// FICTIONAL ENGINEERING PROJECT — NOT FOR CONSTRUCTION
FUNCTION_BLOCK "FB_CellMain"
VAR
   HmiCommands : "FB_HMICommandManager";
   ConveyorVfd : "FB_VFD";
   PumpVfd : "FB_VFD";
   Gate : "FB_Actuator2Pos";
   Clamp : "FB_Actuator2Pos";
   FillCh1 : "FB_FillChannel";
   FillCh2 : "FB_FillChannel";
   Vision : "FB_VisionInterface";
   Capper : "FB_CapperInterface";
   Recipe : "FB_RecipeManager";
   Alarm : "FB_AlarmManager";
   Coordinator : "FB_MachineCoordinator";
   DripTimer : TON;
   PlcHeartbeatTimer : TON;
   blockingFault : Bool;
   outputInterlock : Bool;
   preBlockingFault : Bool;
   immediateStop : Bool;
   processPermissive : Bool;
   modelConfigured : Bool;
   visionOperational : Bool;
   manualConveyorInterlocked : Bool;
   manualSecureInterlocked : Bool;
   manualPumpInterlocked : Bool;
   manualValve1Interlocked : Bool;
   manualValve2Interlocked : Bool;
   activeFaults : Array[0..31] of Bool;
   faultCodes : Array[0..31] of UInt;
   i : Int;
END_VAR
BEGIN
   // Input normalization from process image.
   "DB_IO".Inputs.SafetyOk := %I0.0;
   "DB_IO".Inputs.GuardClosed := %I0.1;
   "DB_IO".Inputs.AirPressureOk := %I0.2;
   "DB_IO".Inputs.ProductSupplyOk := %I0.3;
   "DB_IO".Inputs.Bottle1Present := %I1.2;
   "DB_IO".Inputs.Bottle2Present := %I1.3;
   "DB_IO".Inputs.GateOpen := %I1.4;
   "DB_IO".Inputs.GateClosed := %I1.5;
   "DB_IO".Inputs.ClampReleased := %I1.6;
   "DB_IO".Inputs.ClampEngaged := %I1.7;
   "DB_IO".Inputs.Valve1Closed := %I2.0;
   "DB_IO".Inputs.Valve2Closed := %I2.1;
   "DB_IO".Inputs.CapperReady := %I2.2;
   "DB_IO".Inputs.CapperBusy := %I2.3;
   "DB_IO".Inputs.CapperComplete := %I2.4;
   "DB_IO".Inputs.CapperFault := %I2.5;
   "DB_IO".Inputs.LocalReset := %I2.6;
   "DB_IO".Inputs.LocalStop := %I2.7;
   "DB_IO".Inputs.Flow1Raw := %IW64;
   "DB_IO".Inputs.Flow2Raw := %IW66;
   // Native-project adapter contract. Bind these fields to PN diagnostics and TM Count technology-object outputs in TIA V20.
   "DB_IO".Inputs.ConveyorPnHealthy := "DB_NativeBindings".Inputs.ConveyorPnIoValid;
   "DB_IO".Inputs.PumpPnHealthy := "DB_NativeBindings".Inputs.PumpPnIoValid;
   "DB_IO".Inputs.PulseTotal1 := "DB_NativeBindings".Inputs.Flow1PulseTotal;
   "DB_IO".Inputs.PulseTotal2 := "DB_NativeBindings".Inputs.Flow2PulseTotal;
   "DB_IO".Inputs.Flow1ChannelFault := "DB_NativeBindings".Inputs.Flow1ChannelFault;
   "DB_IO".Inputs.Flow2ChannelFault := "DB_NativeBindings".Inputs.Flow2ChannelFault;
   "DB_IO".Inputs.Flow1PulseChannelFault := "DB_NativeBindings".Inputs.Flow1PulseChannelFault;
   "DB_IO".Inputs.Flow2PulseChannelFault := "DB_NativeBindings".Inputs.Flow2PulseChannelFault;
   "DB_Drives".Conveyor.StatusWord1 := %IW256;
   "DB_Drives".Conveyor.ActualSpeedPzd := %IW258;
   "DB_Drives".Pump.StatusWord1 := %IW260;
   "DB_Drives".Pump.ActualSpeedPzd := %IW262;

   #modelConfigured := "DB_VisionComms".ModelConfigurationApproved AND ("DB_VisionComms".ExpectedModelId <> '') AND (LEN("DB_VisionComms".ExpectedModelHash) = 64)
      AND ("DB_VisionComms".ExpectedDatasetId <> '') AND ("DB_VisionComms".ExpectedCalibrationId <> '')
      AND ("DB_VisionComms".MinimumConfidence > 0.0) AND ("DB_VisionComms".MinimumConfidence <= 1.0)
      AND ("DB_VisionComms".MaximumResultAgeMs > UDINT#0) AND ("DB_VisionComms".MaximumProcessingTimeMs > UDINT#0);
   #visionOperational := "DB_VisionComms".Ready AND "DB_VisionComms".ServiceHealthy AND "DB_VisionComms".CameraHealthy
      AND "DB_VisionComms".ModelLoaded AND NOT "DB_VisionComms".MaintenanceActive;
   #immediateStop := NOT "DB_IO".Inputs.SafetyOk OR NOT "DB_IO".Inputs.GuardClosed OR NOT "DB_IO".Inputs.AirPressureOk OR NOT "DB_IO".Inputs.ProductSupplyOk;
   #processPermissive := NOT #immediateStop AND NOT "DB_IO".PowerRecoveryRequired;
   #preBlockingFault := #immediateStop OR #ConveyorVfd.Fault OR #PumpVfd.Fault OR #Gate.Fault OR #Clamp.Fault OR #FillCh1.Fault OR #FillCh2.Fault OR #Vision.Fault OR NOT #modelConfigured OR NOT #visionOperational OR #Capper.Fault OR NOT #HmiCommands.CommunicationsHealthy;
   #HmiCommands(StartRequest := "DB_HMI".Start.Request, StartSeq := "DB_HMI".Start.RequestSeq, StopRequest := "DB_HMI".ControlledStop.Request, StopSeq := "DB_HMI".ControlledStop.RequestSeq, ResetRequest := "DB_HMI".Reset.Request, ResetSeq := "DB_HMI".Reset.RequestSeq, AckRequest := "DB_HMI".AlarmAck.Request, AckSeq := "DB_HMI".AlarmAck.RequestSeq, AutoRequest := "DB_HMI".AutoMode.Request, AutoSeq := "DB_HMI".AutoMode.RequestSeq, ManualRequest := "DB_HMI".ManualMode.Request, ManualSeq := "DB_HMI".ManualMode.RequestSeq, DispositionRequest := "DB_HMI".DispositionRemoved.Request, DispositionSeq := "DB_HMI".DispositionRemoved.RequestSeq, ManualConveyorRequest := "DB_HMI".ManualConveyorJog.Request, ManualPumpRequest := "DB_HMI".ManualPumpJog.Request, ManualValve1Request := "DB_HMI".ManualValve1.Request, ManualValve2Request := "DB_HMI".ManualValve2.Request, ManualSecureRequest := "DB_HMI".ManualSecure.Request, ManualHoldAllowed := (#Coordinator.State = "E_MachineState".MANUAL_SETUP) AND #processPermissive, LocalStop := "DB_IO".Inputs.LocalStop, LocalReset := "DB_IO".Inputs.LocalReset, CommandHeartbeat := "DB_HMI".CommandHeartbeat, StartAllowed := (#Coordinator.State = "E_MachineState".READY) AND #processPermissive, ResetAllowed := NOT #immediateStop, AutoAllowed := (#Coordinator.State = "E_MachineState".MANUAL_SETUP), ManualAllowed := (#Coordinator.State = "E_MachineState".READY), DispositionAllowed := (#Coordinator.State = "E_MachineState".HOLDING));
   "DB_HMI".Start.AcceptedSeq := #HmiCommands.StartAcceptedSeq; "DB_HMI".Start.RejectedSeq := #HmiCommands.StartRejectedSeq;
   "DB_HMI".ControlledStop.AcceptedSeq := #HmiCommands.StopAcceptedSeq;
   "DB_HMI".Reset.AcceptedSeq := #HmiCommands.ResetAcceptedSeq; "DB_HMI".Reset.RejectedSeq := #HmiCommands.ResetRejectedSeq;
   "DB_HMI".AlarmAck.AcceptedSeq := #HmiCommands.AckAcceptedSeq;
   "DB_HMI".AutoMode.AcceptedSeq := #HmiCommands.AutoAcceptedSeq; "DB_HMI".AutoMode.RejectedSeq := #HmiCommands.AutoRejectedSeq;
   "DB_HMI".ManualMode.AcceptedSeq := #HmiCommands.ManualAcceptedSeq; "DB_HMI".ManualMode.RejectedSeq := #HmiCommands.ManualRejectedSeq;
   "DB_HMI".DispositionRemoved.AcceptedSeq := #HmiCommands.DispositionAcceptedSeq; "DB_HMI".DispositionRemoved.RejectedSeq := #HmiCommands.DispositionRejectedSeq;
   "DB_HMI".CommunicationsHealthy := #HmiCommands.CommunicationsHealthy;
   #manualConveyorInterlocked := #HmiCommands.ManualConveyorCmd AND NOT #HmiCommands.ManualSecureCmd AND NOT #HmiCommands.ManualPumpCmd AND NOT #HmiCommands.ManualValve1Cmd AND NOT #HmiCommands.ManualValve2Cmd AND "DB_IO".Inputs.GateOpen AND "DB_IO".Inputs.ClampReleased;
   #manualSecureInterlocked := #HmiCommands.ManualSecureCmd AND NOT #HmiCommands.ManualConveyorCmd AND #ConveyorVfd.Stopped;
   #manualPumpInterlocked := #HmiCommands.ManualPumpCmd AND #manualSecureInterlocked AND #ConveyorVfd.Stopped AND "DB_IO".Inputs.GateClosed AND "DB_IO".Inputs.ClampEngaged AND (#HmiCommands.ManualValve1Cmd OR #HmiCommands.ManualValve2Cmd);
   #manualValve1Interlocked := #HmiCommands.ManualValve1Cmd AND #manualPumpInterlocked AND #PumpVfd.Running;
   #manualValve2Interlocked := #HmiCommands.ManualValve2Cmd AND #manualPumpInterlocked AND #PumpVfd.Running;
   "DB_HMI".Start.Allowed := (#Coordinator.State = "E_MachineState".READY) AND #processPermissive; "DB_HMI".Start.Busy := FALSE; "DB_HMI".Start.DisabledReason := 0; IF NOT "DB_HMI".Start.Allowed THEN "DB_HMI".Start.DisabledReason := 1; END_IF;
   "DB_HMI".ControlledStop.Allowed := TRUE; "DB_HMI".ControlledStop.Busy := FALSE; "DB_HMI".ControlledStop.DisabledReason := 0;
   "DB_HMI".Reset.Allowed := NOT #immediateStop; "DB_HMI".Reset.Busy := FALSE; "DB_HMI".Reset.DisabledReason := 0; IF NOT "DB_HMI".Reset.Allowed THEN "DB_HMI".Reset.DisabledReason := 2; END_IF;
   "DB_HMI".AlarmAck.Allowed := TRUE; "DB_HMI".AlarmAck.Busy := FALSE; "DB_HMI".AlarmAck.DisabledReason := 0;
   "DB_HMI".AutoMode.Allowed := (#Coordinator.State = "E_MachineState".MANUAL_SETUP); "DB_HMI".AutoMode.Busy := FALSE; "DB_HMI".AutoMode.DisabledReason := 0; IF NOT "DB_HMI".AutoMode.Allowed THEN "DB_HMI".AutoMode.DisabledReason := 4; END_IF;
   "DB_HMI".ManualMode.Allowed := (#Coordinator.State = "E_MachineState".READY); "DB_HMI".ManualMode.Busy := FALSE; "DB_HMI".ManualMode.DisabledReason := 0; IF NOT "DB_HMI".ManualMode.Allowed THEN "DB_HMI".ManualMode.DisabledReason := 4; END_IF;
   "DB_HMI".DispositionRemoved.Allowed := (#Coordinator.State = "E_MachineState".HOLDING); "DB_HMI".DispositionRemoved.Busy := FALSE; "DB_HMI".DispositionRemoved.DisabledReason := 0;
   "DB_HMI".ManualConveyorJog.Allowed := (#Coordinator.State = "E_MachineState".MANUAL_SETUP) AND #processPermissive AND NOT #HmiCommands.ManualSecureCmd AND NOT #HmiCommands.ManualPumpCmd AND NOT #HmiCommands.ManualValve1Cmd AND NOT #HmiCommands.ManualValve2Cmd AND "DB_IO".Inputs.GateOpen AND "DB_IO".Inputs.ClampReleased; "DB_HMI".ManualConveyorJog.Busy := #manualConveyorInterlocked; "DB_HMI".ManualConveyorJog.DisabledReason := 0; IF NOT "DB_HMI".ManualConveyorJog.Allowed THEN "DB_HMI".ManualConveyorJog.DisabledReason := 5; END_IF;
   "DB_HMI".ManualPumpJog.Allowed := (#Coordinator.State = "E_MachineState".MANUAL_SETUP) AND #processPermissive AND #manualSecureInterlocked AND #ConveyorVfd.Stopped AND "DB_IO".Inputs.GateClosed AND "DB_IO".Inputs.ClampEngaged; "DB_HMI".ManualPumpJog.Busy := #manualPumpInterlocked; "DB_HMI".ManualPumpJog.DisabledReason := 0; IF NOT "DB_HMI".ManualPumpJog.Allowed THEN "DB_HMI".ManualPumpJog.DisabledReason := 6; END_IF;
   "DB_HMI".ManualValve1.Allowed := "DB_HMI".ManualPumpJog.Allowed; "DB_HMI".ManualValve1.Busy := #manualValve1Interlocked; "DB_HMI".ManualValve1.DisabledReason := "DB_HMI".ManualPumpJog.DisabledReason;
   "DB_HMI".ManualValve2.Allowed := "DB_HMI".ManualPumpJog.Allowed; "DB_HMI".ManualValve2.Busy := #manualValve2Interlocked; "DB_HMI".ManualValve2.DisabledReason := "DB_HMI".ManualPumpJog.DisabledReason;
   "DB_HMI".ManualSecure.Allowed := (#Coordinator.State = "E_MachineState".MANUAL_SETUP) AND #processPermissive AND #ConveyorVfd.Stopped AND NOT #HmiCommands.ManualConveyorCmd; "DB_HMI".ManualSecure.Busy := #manualSecureInterlocked; "DB_HMI".ManualSecure.DisabledReason := 0; IF NOT "DB_HMI".ManualSecure.Allowed THEN "DB_HMI".ManualSecure.DisabledReason := 7; END_IF;

   #Recipe(Candidate := "DB_Recipe".Candidate, ApplyRequest := "DB_HMI".RecipeApply.Request AND #HmiCommands.CommunicationsHealthy, RequestSeq := "DB_HMI".RecipeApply.RequestSeq, MachineStopped := (#Coordinator.State = "E_MachineState".STOPPED));
   "DB_Recipe".Active := #Recipe.Active;
   "DB_HMI".RecipeApply.AcceptedSeq := #Recipe.AcceptedSeq; "DB_HMI".RecipeApply.RejectedSeq := #Recipe.RejectedSeq;
   "DB_HMI".RecipeApply.Allowed := (#Coordinator.State = "E_MachineState".STOPPED) AND #Recipe.Valid; "DB_HMI".RecipeApply.Busy := FALSE; "DB_HMI".RecipeApply.DisabledReason := 0; IF NOT #Recipe.Valid THEN "DB_HMI".RecipeApply.DisabledReason := 3; END_IF;

   "DB_Drives".Conveyor.CommsHealthy := "DB_IO".Inputs.ConveyorPnHealthy; "DB_Drives".Pump.CommsHealthy := "DB_IO".Inputs.PumpPnHealthy;
   #ConveyorVfd(Enable := "DB_IO".Inputs.SafetyOk AND "DB_IO".Inputs.GuardClosed, RunRequest := (#Coordinator.IndexRequest OR #manualConveyorInterlocked) AND NOT #immediateStop, ResetEdge := #HmiCommands.ResetPulse, CommsHealthy := "DB_Drives".Conveyor.CommsHealthy, StatusWord1 := "DB_Drives".Conveyor.StatusWord1, ActualSpeedPzd := "DB_Drives".Conveyor.ActualSpeedPzd, SpeedReferencePct := 35.0, StartTimeout := T#3s, StopTimeout := T#3s);
   #PumpVfd(Enable := #processPermissive, RunRequest := ((#FillCh1.PumpRequest OR #FillCh2.PumpRequest) OR #manualPumpInterlocked) AND #processPermissive, ResetEdge := #HmiCommands.ResetPulse, CommsHealthy := "DB_Drives".Pump.CommsHealthy, StatusWord1 := "DB_Drives".Pump.StatusWord1, ActualSpeedPzd := "DB_Drives".Pump.ActualSpeedPzd, SpeedReferencePct := 60.0, StartTimeout := T#3s, StopTimeout := T#3s);
   "DB_Drives".Conveyor.Ready := #ConveyorVfd.Ready; "DB_Drives".Conveyor.Running := #ConveyorVfd.Running; "DB_Drives".Conveyor.Fault := #ConveyorVfd.Fault; "DB_Drives".Conveyor.ActualSpeedPct := #ConveyorVfd.ActualSpeedPct;
   "DB_Drives".Pump.Ready := #PumpVfd.Ready; "DB_Drives".Pump.Running := #PumpVfd.Running; "DB_Drives".Pump.Fault := #PumpVfd.Fault; "DB_Drives".Pump.ActualSpeedPct := #PumpVfd.ActualSpeedPct;
   #Gate(Enable := NOT #immediateStop, CmdToA := NOT (#Coordinator.GateCloseRequest OR #manualSecureInterlocked), CmdToB := #Coordinator.GateCloseRequest OR #manualSecureInterlocked, AtA := "DB_IO".Inputs.GateOpen, AtB := "DB_IO".Inputs.GateClosed, ResetEdge := #HmiCommands.ResetPulse, TravelTime := T#2s);
   #Clamp(Enable := NOT #immediateStop, CmdToA := NOT (#Coordinator.ClampRequest OR #manualSecureInterlocked), CmdToB := #Coordinator.ClampRequest OR #manualSecureInterlocked, AtA := "DB_IO".Inputs.ClampReleased, AtB := "DB_IO".Inputs.ClampEngaged, ResetEdge := #HmiCommands.ResetPulse, TravelTime := T#2s);
   #FillCh1(Enable := #processPermissive, PumpRunning := #PumpVfd.Running, StartEdge := #Coordinator.FillStartPulse, Abort := #preBlockingFault OR #ConveyorVfd.Fault OR #PumpVfd.Fault OR #Gate.Fault OR #Clamp.Fault OR #HmiCommands.StopPulse, ResetEdge := #HmiCommands.ResetPulse, PulseTotal := "DB_IO".Inputs.PulseTotal1, FlowRaw := "DB_IO".Inputs.Flow1Raw, PulseChannelFault := "DB_IO".Inputs.Flow1PulseChannelFault, AnalogChannelFault := "DB_IO".Inputs.Flow1ChannelFault, ValveClosedFb := "DB_IO".Inputs.Valve1Closed, TargetMl := "DB_Recipe".Active.TargetMlCh1, PulsesPerLitre := "DB_Recipe".Active.PulsesPerLitreCh1, UnderToleranceMl := "DB_Recipe".Active.UnderToleranceMl, OverToleranceMl := "DB_Recipe".Active.OverToleranceMl, FlowMaxLMin := 20.0, NoFlowMinLMin := 0.2, PlausibilityPct := 25.0, PulseWindowTimeS := "DB_Recipe".Active.PulseWindowTimeS, NoFlowTimeout := "DB_Recipe".Active.NoFlowTimeout, FillTimeout := "DB_Recipe".Active.FillTimeout, ValveOpenTimeout := "DB_Recipe".Active.ValveOpenTimeout, ValveCloseTimeout := "DB_Recipe".Active.ValveCloseTimeout, PlausibilityTime := "DB_Recipe".Active.PlausibilityTime);
   #FillCh2(Enable := #processPermissive, PumpRunning := #PumpVfd.Running, StartEdge := #Coordinator.FillStartPulse, Abort := #preBlockingFault OR #ConveyorVfd.Fault OR #PumpVfd.Fault OR #Gate.Fault OR #Clamp.Fault OR #HmiCommands.StopPulse, ResetEdge := #HmiCommands.ResetPulse, PulseTotal := "DB_IO".Inputs.PulseTotal2, FlowRaw := "DB_IO".Inputs.Flow2Raw, PulseChannelFault := "DB_IO".Inputs.Flow2PulseChannelFault, AnalogChannelFault := "DB_IO".Inputs.Flow2ChannelFault, ValveClosedFb := "DB_IO".Inputs.Valve2Closed, TargetMl := "DB_Recipe".Active.TargetMlCh2, PulsesPerLitre := "DB_Recipe".Active.PulsesPerLitreCh2, UnderToleranceMl := "DB_Recipe".Active.UnderToleranceMl, OverToleranceMl := "DB_Recipe".Active.OverToleranceMl, FlowMaxLMin := 20.0, NoFlowMinLMin := 0.2, PlausibilityPct := 25.0, PulseWindowTimeS := "DB_Recipe".Active.PulseWindowTimeS, NoFlowTimeout := "DB_Recipe".Active.NoFlowTimeout, FillTimeout := "DB_Recipe".Active.FillTimeout, ValveOpenTimeout := "DB_Recipe".Active.ValveOpenTimeout, ValveCloseTimeout := "DB_Recipe".Active.ValveCloseTimeout, PlausibilityTime := "DB_Recipe".Active.PlausibilityTime);
   #DripTimer(IN := (#Coordinator.AutoStep = "E_AutoStep".DRIP_SETTLE), PT := "DB_Recipe".Active.DripSettleTime);
   #Capper(Enable := NOT #immediateStop, RequestEdge := #Coordinator.CapperRequestPulse, Ready := "DB_IO".Inputs.CapperReady, Busy := "DB_IO".Inputs.CapperBusy, Complete := "DB_IO".Inputs.CapperComplete, FaultIn := "DB_IO".Inputs.CapperFault, ResetEdge := #HmiCommands.ResetPulse, AcceptTimeout := T#2s, CompleteTimeout := T#10s);
   // Allocate exactly one immutable ID. A repeated coordinator pulse cannot mutate
   // the externally visible transaction while the vision interface is pending.
   IF #Coordinator.VisionRequestPulse AND NOT #Vision.RequestInProgress AND ("DB_VisionComms".InspectionId < UDINT#4294967295) THEN "DB_VisionComms".InspectionId := "DB_VisionComms".InspectionId + UDINT#1; END_IF;
   // READY low holds VISION_ENABLE low so a cold/restarted edge can atomically
   // seed the PLC session/ID/ACK/heartbeat snapshot before declaring READY.
   "DB_VisionComms".MaintenanceMode := (#Coordinator.State = "E_MachineState".MANUAL_SETUP);
   "DB_VisionComms".Enable := #processPermissive AND #modelConfigured AND "DB_VisionComms".Ready AND #visionOperational
      AND NOT "DB_VisionComms".MaintenanceMode AND NOT #Vision.Fault;
   "DB_VisionComms".RecipeId := "DB_Recipe".Active.RecipeId; "DB_VisionComms".ExpectedBottles := 2; "DB_VisionComms".TargetFillLevel := "DB_Recipe".Active.TargetFillLevel;
   #PlcHeartbeatTimer(IN := NOT #PlcHeartbeatTimer.Q, PT := T#500ms);
   IF #PlcHeartbeatTimer.Q THEN
      IF "DB_VisionComms".PlcHeartbeat = UDINT#4294967295 THEN "DB_VisionComms".PlcHeartbeat := UDINT#0;
      ELSE "DB_VisionComms".PlcHeartbeat := "DB_VisionComms".PlcHeartbeat + UDINT#1; END_IF;
   END_IF;
   #Vision(Enable := "DB_VisionComms".Enable, TriggerEdge := #Coordinator.VisionRequestPulse,
      InspectionId := "DB_VisionComms".InspectionId, SessionEpoch := "DB_VisionComms".SessionEpoch,
      ExpectedModelId := "DB_VisionComms".ExpectedModelId, ExpectedModelHash := "DB_VisionComms".ExpectedModelHash,
      ExpectedDatasetId := "DB_VisionComms".ExpectedDatasetId, ExpectedCalibrationId := "DB_VisionComms".ExpectedCalibrationId,
      MinimumConfidence := "DB_VisionComms".MinimumConfidence, MaximumResultAgeMs := "DB_VisionComms".MaximumResultAgeMs,
      MaximumProcessingTimeMs := "DB_VisionComms".MaximumProcessingTimeMs, MaximumQueueDepth := "DB_VisionComms".MaximumQueueDepth,
      Ready := "DB_VisionComms".Ready, Busy := "DB_VisionComms".Busy, CaptureAckId := "DB_VisionComms".CaptureAckId,
      ProcessingState := "DB_VisionComms".ProcessingState, ServiceHealthy := "DB_VisionComms".ServiceHealthy,
      CameraHealthy := "DB_VisionComms".CameraHealthy, ModelLoaded := "DB_VisionComms".ModelLoaded,
      MaintenanceActive := "DB_VisionComms".MaintenanceActive, QueueDepth := "DB_VisionComms".QueueDepth,
      Result := "DB_VisionComms".Result, Heartbeat := "DB_VisionComms".VisionHeartbeat,
      Timeout := "DB_Recipe".Active.VisionTimeout, HeartbeatTimeout := T#1s, ResetEdge := #HmiCommands.ResetPulse);
   "DB_VisionComms".Trigger := #Vision.Trigger;
   "DB_VisionComms".ResultAgeMs := #Vision.ResultAgeMs;
   IF NOT #modelConfigured THEN "DB_VisionComms".DiagReason := "E_VisionDiag".MODEL_MISMATCH;
   ELSIF NOT "DB_VisionComms".ServiceHealthy THEN "DB_VisionComms".DiagReason := "E_VisionDiag".SERVICE_UNHEALTHY;
   ELSIF NOT "DB_VisionComms".CameraHealthy THEN "DB_VisionComms".DiagReason := "E_VisionDiag".CAMERA_UNHEALTHY;
   ELSIF NOT "DB_VisionComms".ModelLoaded THEN "DB_VisionComms".DiagReason := "E_VisionDiag".MODEL_NOT_LOADED;
   ELSIF "DB_VisionComms".MaintenanceActive THEN "DB_VisionComms".DiagReason := "E_VisionDiag".MAINTENANCE_ACTIVE;
   ELSE "DB_VisionComms".DiagReason := #Vision.DiagReason; END_IF;
   IF #Vision.PublicationAck THEN "DB_VisionComms".ResultAckId := "DB_VisionComms".Result.ResultId; END_IF;
   FOR #i := 0 TO 31 DO #activeFaults[#i] := FALSE; #faultCodes[#i] := 0; END_FOR;
   #activeFaults[0] := NOT "DB_IO".Inputs.SafetyOk; #faultCodes[0] := 1001;
   #activeFaults[1] := NOT "DB_IO".Inputs.GuardClosed; #faultCodes[1] := 1004;
   #activeFaults[2] := NOT "DB_IO".Inputs.AirPressureOk; #faultCodes[2] := 1002;
   #activeFaults[3] := NOT "DB_IO".Inputs.ProductSupplyOk; #faultCodes[3] := 1003;
   #activeFaults[4] := #ConveyorVfd.Fault; #faultCodes[4] := 1101;
   #activeFaults[5] := #PumpVfd.Fault; #faultCodes[5] := 1102;
   #activeFaults[6] := #Gate.Fault; #faultCodes[6] := 1201;
   #activeFaults[7] := #Clamp.Fault; #faultCodes[7] := 1202;
   #activeFaults[8] := #FillCh1.Fault; CASE #FillCh1.DiagReason OF "E_FillDiag".ANALOG_BROKEN_WIRE: #faultCodes[8] := 1307; "E_FillDiag".NO_FLOW: #faultCodes[8] := 1301; "E_FillDiag".PULSE_MISSING: #faultCodes[8] := 1321; "E_FillDiag".ANALOG_NO_FLOW: #faultCodes[8] := 1322; "E_FillDiag".PULSE_ANALOG_DISAGREE: #faultCodes[8] := 1303; "E_FillDiag".UNDERFILL: #faultCodes[8] := 1304; "E_FillDiag".OVERFILL: #faultCodes[8] := 1305; "E_FillDiag".VALVE_OPEN_MISMATCH: #faultCodes[8] := 1308; "E_FillDiag".VALVE_CLOSE_MISMATCH: #faultCodes[8] := 1306; "E_FillDiag".CONTINUED_FLOW: #faultCodes[8] := 1309; ELSE #faultCodes[8] := 1310; END_CASE;
   #activeFaults[9] := #FillCh2.Fault; CASE #FillCh2.DiagReason OF "E_FillDiag".ANALOG_BROKEN_WIRE: #faultCodes[9] := 1317; "E_FillDiag".NO_FLOW: #faultCodes[9] := 1311; "E_FillDiag".PULSE_MISSING: #faultCodes[9] := 1323; "E_FillDiag".ANALOG_NO_FLOW: #faultCodes[9] := 1324; "E_FillDiag".PULSE_ANALOG_DISAGREE: #faultCodes[9] := 1313; "E_FillDiag".UNDERFILL: #faultCodes[9] := 1314; "E_FillDiag".OVERFILL: #faultCodes[9] := 1315; "E_FillDiag".VALVE_OPEN_MISMATCH: #faultCodes[9] := 1318; "E_FillDiag".VALVE_CLOSE_MISMATCH: #faultCodes[9] := 1316; "E_FillDiag".CONTINUED_FLOW: #faultCodes[9] := 1319; ELSE #faultCodes[9] := 1320; END_CASE;
   #activeFaults[10] := #Vision.Fault OR #Vision.HoldRequired OR NOT #modelConfigured OR NOT "DB_VisionComms".Ready;
   #activeFaults[10] := #activeFaults[10] OR NOT #visionOperational;
   IF NOT #modelConfigured THEN #faultCodes[10] := 1506;
   ELSIF NOT "DB_VisionComms".Ready AND NOT #Vision.Fault AND NOT #Vision.HoldRequired THEN #faultCodes[10] := 1501;
   ELSE CASE #Vision.DiagReason OF "E_VisionDiag".READY_TIMEOUT: #faultCodes[10] := 1501; "E_VisionDiag".RESULT_TIMEOUT: #faultCodes[10] := 1502; "E_VisionDiag".RESULT_ID_MISMATCH: #faultCodes[10] := 1503; "E_VisionDiag".QUALITY_BLOCK: #faultCodes[10] := 1504; "E_VisionDiag".HEARTBEAT_LOSS: #faultCodes[10] := 1505; ELSE #faultCodes[10] := 1506; END_CASE; END_IF;
   #activeFaults[11] := #Capper.Fault; IF (#Capper.DiagReason = 1) OR (#Capper.DiagReason = 5) THEN #faultCodes[11] := 1402; ELSE #faultCodes[11] := 1401; END_IF;
   #activeFaults[12] := NOT #HmiCommands.CommunicationsHealthy; #faultCodes[12] := 1601;
   // Quality holds remain alarmed and output-interlocked but are not equipment
   // faults; this preserves the coordinator's INSPECT -> HOLDING disposition path.
   #blockingFault := #immediateStop OR #ConveyorVfd.Fault OR #PumpVfd.Fault OR #Gate.Fault OR #Clamp.Fault OR #FillCh1.Fault OR #FillCh2.Fault OR #Vision.Fault OR NOT #modelConfigured OR NOT "DB_VisionComms".Ready OR NOT #visionOperational OR #Capper.Fault OR NOT #HmiCommands.CommunicationsHealthy;
   // A restart never reprocesses a bottle already in the cell. Recovery is
   // acknowledged only after the cell is physically empty.
   IF #HmiCommands.ResetPulse AND NOT #blockingFault AND NOT "DB_IO".Inputs.Bottle1Present AND NOT "DB_IO".Inputs.Bottle2Present THEN "DB_IO".PowerRecoveryRequired := FALSE; #processPermissive := NOT #immediateStop; END_IF;
   #Coordinator(InitDone := TRUE, PermissivesOk := #processPermissive, StartEdge := #HmiCommands.StartPulse, StopEdge := #HmiCommands.StopPulse, ResetEdge := #HmiCommands.ResetPulse, AutoRequest := #HmiCommands.AutoPulse, ManualRequest := #HmiCommands.ManualPulse, DispositionRemoved := #HmiCommands.DispositionPulse, PairPresent := "DB_IO".Inputs.Bottle1Present AND "DB_IO".Inputs.Bottle2Present, PairAbsent := NOT "DB_IO".Inputs.Bottle1Present AND NOT "DB_IO".Inputs.Bottle2Present, ConveyorStopped := #ConveyorVfd.Stopped, GateClosed := "DB_IO".Inputs.GateClosed, GateOpen := "DB_IO".Inputs.GateOpen, ClampEngaged := "DB_IO".Inputs.ClampEngaged, ClampReleased := "DB_IO".Inputs.ClampReleased, Fill1Done := #FillCh1.Done, Fill2Done := #FillCh2.Done, DripDone := #DripTimer.Q, VisionAccepted := #Vision.Accepted, VisionPass := #Vision.QualityPass, CapperReady := "DB_IO".Inputs.CapperReady, CapperComplete := #Capper.CompletePulse, BlockingFault := #blockingFault);
   #Alarm(ActiveFaults := #activeFaults, FaultCodes := #faultCodes, AckEdge := #HmiCommands.AckPulse, ResetEdge := #HmiCommands.ResetPulse);
   "DB_HMI".FirstOutAlarm := #Alarm.FirstOutCode;

   // Final physical-output mapping. HMI never writes this structure.
   #outputInterlock := #blockingFault OR #Vision.HoldRequired OR #Coordinator.QualityHold;
   "DB_IO".ReleasePermissive := #processPermissive AND NOT #outputInterlock;
   "DB_IO".Commands.FillValve1 := (#FillCh1.ValveOpenCmd OR #manualValve1Interlocked) AND "DB_IO".ReleasePermissive;
   "DB_IO".Commands.FillValve2 := (#FillCh2.ValveOpenCmd OR #manualValve2Interlocked) AND "DB_IO".ReleasePermissive;
   "DB_IO".Commands.GateOpen := #Gate.OutToA AND "DB_IO".ReleasePermissive;
   "DB_IO".Commands.GateClose := #Gate.OutToB AND "DB_IO".ReleasePermissive;
   "DB_IO".Commands.ClampRelease := #Clamp.OutToA AND "DB_IO".ReleasePermissive;
   "DB_IO".Commands.ClampEngage := #Clamp.OutToB AND "DB_IO".ReleasePermissive;
   "DB_IO".Commands.CapperRequest := #Capper.Request AND "DB_IO".ReleasePermissive;
   "DB_IO".Commands.CameraLight := (#Coordinator.AutoStep = "E_AutoStep".INSPECT) AND "DB_IO".ReleasePermissive;
   "DB_IO".Commands.StackGreen := (#Coordinator.State = "E_MachineState".AUTOMATIC) AND NOT #outputInterlock;
   "DB_IO".Commands.StackAmber := (#Coordinator.State = "E_MachineState".HOLDING) OR (#Coordinator.State = "E_MachineState".MANUAL_SETUP);
   "DB_IO".Commands.StackRed := #blockingFault; "DB_IO".Commands.Audible := #Alarm.AnyFault AND NOT #Alarm.Acknowledged;
   %Q0.2 := "DB_IO".Commands.FillValve1; %Q0.3 := "DB_IO".Commands.FillValve2;
   %Q0.4 := "DB_IO".Commands.GateOpen; %Q0.5 := "DB_IO".Commands.GateClose;
   %Q0.6 := "DB_IO".Commands.ClampEngage; %Q0.7 := "DB_IO".Commands.ClampRelease;
   %Q1.0 := "DB_IO".Commands.CapperRequest;
   %Q1.1 := "DB_IO".Commands.StackGreen; %Q1.2 := "DB_IO".Commands.StackAmber; %Q1.3 := "DB_IO".Commands.StackRed; %Q1.4 := "DB_IO".Commands.Audible; %Q1.5 := "DB_IO".Commands.CameraLight;
   IF "DB_IO".ReleasePermissive THEN %QW256 := #ConveyorVfd.ControlWord1; %QW258 := #ConveyorVfd.SpeedSetpointPzd; %QW260 := #PumpVfd.ControlWord1; %QW262 := #PumpVfd.SpeedSetpointPzd;
   ELSE %QW256 := W#16#047E; %QW258 := 0; %QW260 := W#16#047E; %QW262 := 0; END_IF;
   "DB_HMI".StateCode := ENUM_TO_UINT(#Coordinator.State); "DB_HMI".AutoStepCode := ENUM_TO_UINT(#Coordinator.AutoStep); "DB_HMI".QualityHold := #Coordinator.QualityHold OR #Coordinator.DispositionRequired;
END_FUNCTION_BLOCK
